Yaskawa INFORM job: TWIN_FRONT_WELD_-90ST-1_5340.JBI

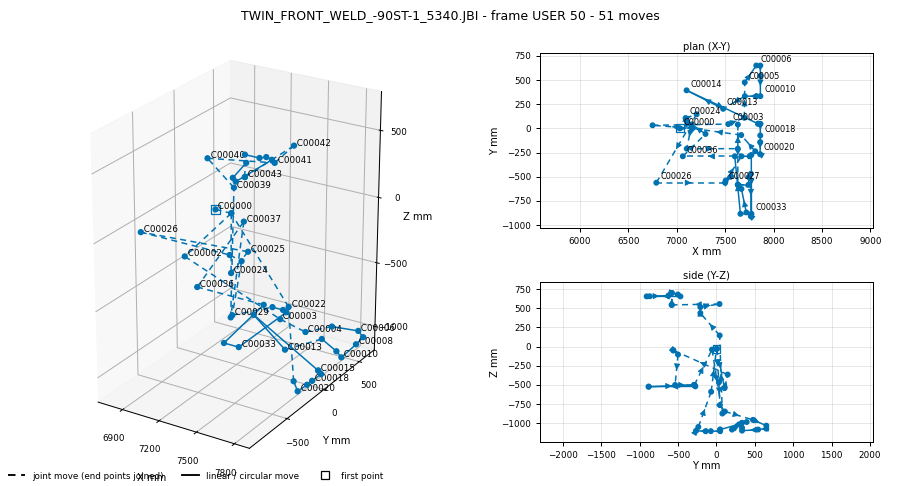
[picture p0: tool path of TWIN_FRONT_WELD_-90ST-1_5340.JBI in frame USER 50, 51 of 52 moves have a stored position in this frame; points joined in program order, loops and branches not executed]
/JOB
//NAME TWIN_FRONT_WELD_-90ST-1_5340
///FOLDERNAME 02-SKRZYNIE_JOBS
//POS
///NPOS 52,52,0,8,0,0
///USER 50
///TOOL 0
///POSTYPE USER
///RECTAN
///RCONF 0,0,1,0,0,0,0,0,0,0,0,0,0,0,0,0,0,0,0,0,0,0,0,0
C00000=7029.164,0.308,-30.113,-0.0036,-53.6521,0.0034
C00001=7158.107,0.312,-30.113,0.0036,-53.6521,-0.0034
///RCONF 1,0,1,0,0,0,0,0,0,0,0,0,0,0,0,0,0,0,0,0,0,0,0,0
C00002=6749.002,31.739,-465.549,-15.1595,35.6819,145.6807
///RCONF 1,0,0,0,0,0,0,0,0,0,0,0,0,0,0,0,0,0,0,0,0,0,0,0
C00003=7531.423,44.323,-762.797,-8.7291,34.6461,164.2133
C00004=7698.038,109.341,-845.576,-15.9625,40.0165,157.0814
C00005=7701.880,475.670,-954.346,-13.0495,30.7936,159.1476
C00006=7821.278,649.645,-1029.983,-23.6743,36.9906,149.9805
C00007=7862.724,649.337,-1069.296,-23.6733,36.9909,149.9831
C00008=7864.081,542.033,-1080.239,-23.6771,36.9818,149.9803
C00009=7863.681,455.675,-1087.596,-23.6808,36.9789,149.9684
C00010=7863.526,332.886,-1094.548,-23.6820,36.9781,149.9731
C00011=7822.668,332.804,-1057.389,-23.6776,36.9789,149.9852
C00012=7702.743,332.795,-992.444,-23.6771,36.9773,149.9828
C00013=7478.605,202.215,-1080.996,-5.5877,19.7754,112.8961
C00014=7100.516,393.258,-982.274,31.5072,20.3423,57.1288
///RCONF 0,0,0,0,0,0,0,0,0,0,0,0,0,0,0,0,0,0,0,0,0,0,0,0
C00015=7840.287,47.964,-1081.198,-15.4598,43.5968,152.6291
C00016=7840.287,47.964,-1081.198,-15.4598,43.5968,152.6291
C00017=7863.996,47.345,-1101.690,-15.0733,42.7558,153.1362
C00018=7862.274,-73.558,-1101.821,-15.0685,42.7518,153.1415
C00019=7862.125,-142.007,-1102.138,-15.0642,42.7510,153.1502
C00020=7860.827,-266.961,-1097.466,-11.5759,45.8640,155.5433
C00021=7810.369,-236.945,-1047.165,-12.8910,39.7294,154.3361
C00022=7665.368,-69.314,-588.357,-56.5185,9.2692,73.1107
///RCONF 0,0,1,0,0,0,0,0,0,0,0,0,0,0,0,0,0,0,0,0,0,0,0,0
C00023=7158.107,0.312,-30.113,0.0036,-53.6521,-0.0034
///RCONF 1,0,0,0,0,0,0,0,0,0,0,0,0,0,0,0,0,0,0,0,0,0,0,0
C00024=7089.632,105.235,-540.772,34.6747,-14.1850,-36.1511
///RCONF 0,0,0,0,0,0,0,0,0,0,0,0,0,0,0,0,0,0,0,0,0,0,0,0
C00025=7204.424,145.895,-364.343,71.1061,41.6311,-75.1821
///RCONF 1,0,1,0,0,0,0,0,0,0,0,0,0,0,0,0,0,0,0,0,0,0,0,0
C00026=6787.828,-561.979,-49.248,-84.3346,30.5101,20.5434
///RCONF 0,0,1,0,1,0,0,0,0,0,0,0,0,0,0,0,0,0,0,0,0,0,0,0
C00027=7499.847,-561.979,-49.248,-84.3345,30.5096,20.5433
///RCONF 0,0,1,0,0,0,0,0,0,0,0,0,0,0,0,0,0,0,0,0,0,0,0,0
C00028=7554.743,-500.998,-104.255,54.0039,-31.4868,-103.9439
///RCONF 0,0,0,0,0,0,0,0,0,0,0,0,0,0,0,0,0,0,0,0,0,0,0,0
C00029=7504.887,-539.129,-499.841,26.1477,-33.6094,-90.8544
C00030=7668.096,-288.720,-499.869,26.1496,-33.6072,-90.8555
C00031=7751.665,-288.695,-499.888,50.2103,-29.8101,-103.4316
C00032=7769.646,-275.360,-518.298,50.1633,-29.8093,-103.3948
C00033=7771.403,-883.462,-522.090,50.1989,-29.8077,-103.4313
C00034=7657.159,-883.464,-522.091,50.1980,-29.8087,-103.4305
C00035=7598.862,-288.695,-499.888,50.2103,-29.8101,-103.4316
C00036=7061.929,-288.695,-499.888,50.2103,-29.8101,-103.4316
C00037=7296.409,-57.933,-39.561,132.2856,-81.6072,-138.1355
C00038=7103.855,76.465,-871.663,11.0010,-20.3154,-11.3718
///RCONF 1,0,1,0,0,0,0,0,0,0,0,0,0,0,0,0,0,0,0,0,0,0,0,0
C00039=7154.189,41.489,145.490,17.6136,-33.4406,-10.5318
C00040=7102.089,-209.900,436.597,-19.7303,-44.5925,9.1969
C00041=7630.528,-209.897,514.987,-19.7320,-44.5912,9.1993
C00042=7630.530,39.680,554.688,-52.1357,-35.3916,30.4208
C00043=7630.500,-582.850,542.955,-61.9434,-30.0005,35.7331
C00044=7630.491,-582.857,542.952,-61.9449,-29.9979,35.7338
C00045=7630.501,-582.856,698.927,-61.9436,-29.9977,35.7338
C00046=7740.859,-582.856,698.927,-61.9436,-29.9977,35.7338
C00047=7743.607,-503.312,679.062,-61.9419,-29.9985,35.7328
C00048=7765.899,-469.746,653.450,-60.1061,-26.9469,34.8664
C00049=7765.598,-909.634,654.025,-56.0408,-31.7443,29.4745
C00050=7718.203,-868.976,655.452,-56.0446,-31.7378,29.4783
C00051=7667.415,-626.051,664.446,-58.3119,-31.1539,31.9267
///RCONF 0,0,0,0,0,0,0,0,0,0,0,0,0,0,0,0,0,0,0,0,0,0,0,0
BC00000=5214.746
BC00001=5343.689
BC00002=5343.689
BC00003=6178.800
BC00004=6495.017
BC00005=6648.627
BC00006=6688.143
BC00007=6688.143
BC00008=6688.143
BC00009=6688.144
BC00010=6688.144
BC00011=6688.143
BC00012=6688.143
BC00013=6688.144
BC00014=6688.143
BC00015=6686.021
BC00016=6686.021
BC00017=6686.021
BC00018=6686.034
BC00019=6686.047
BC00020=6686.060
BC00021=6686.021
BC00022=6015.470
BC00023=5343.689
BC00024=5388.459
BC00025=5388.459
BC00026=5388.459
BC00027=6100.478
BC00028=6100.478
BC00029=6331.805
BC00030=6331.805
BC00031=6331.805
BC00032=6331.785
BC00033=6331.785
BC00034=6331.785
BC00035=6179.002
BC00036=5642.069
BC00037=5642.069
BC00038=5642.069
BC00039=5642.069
BC00040=5642.069
BC00041=6170.513
BC00042=6170.513
BC00043=6170.513
BC00044=6302.692
BC00045=6302.692
BC00046=6413.050
BC00047=6413.050
BC00048=6413.056
BC00049=6735.412
BC00050=6672.519
BC00051=6394.301
///POSTYPE BASE
P00021=6.550,-0.003,-5.735,0.0000,0.0000,0.0000
P00022=5.943,-0.018,-6.388,0.0000,0.0000,0.0000
P00023=7.025,-0.019,-7.168,0.0000,0.0000,0.0000
P00024=5.926,-0.047,-4.777,0.0000,0.0000,0.0000
P00501=-2.026,0.009,3.534,0.0000,0.0000,0.0000
///RCONF 1,0,0,0,0,0,0,0,0,0,0,0,0,0,0,0,0,0,0,0,0,0,0,0
P00502=-2.023,0.001,1.732,0.0000,0.0000,0.0000
P00503=0.138,-0.044,1.539,0.0000,0.0000,0.0000
P00504=-0.309,-0.010,1.636,0.0000,0.0000,0.0000
//INST
///DATE 2024/12/18 13:42
///ATTR SC,RW,RJ
////FRAME USER 50
///GROUP1 RB1,BS1
NOP
MOVJ C00000 BC00000 VJ=50.00
MOVJ C00001 BC00001 VJ=50.00
MOVJ C00002 BC00002 VJ=50.00
MOVJ C00003 BC00003 VJ=50.00
MOVJ C00004 BC00004 VJ=50.00
MOVJ C00005 BC00005 VJ=50.00
'::::::::::::::::::::::::::::::::
'W56
'::::::::::::::::::::::::::::::::
MOVL C00006 BC00006 V=500.0
SFTON P0501
MACRO1 MJ#(0) ARGF14
MOVL C00007 BC00007 V=166.7 PL=0
ARCON
MOVC C00008 BC00008 V=9.5
SFTOF
SFTON P0502
MOVC C00009 BC00009 V=9.5
MOVC C00010 BC00010 V=9.5
ARCOF
MOVL C00011 BC00011 V=166.7
SFTOF
MOVL C00012 BC00012 V=166.7
MOVJ C00013 BC00013 VJ=30.00
MOVL C00014 BC00014 V=166.7
MOVL C00015 BC00015 V=166.7
'::::::::::::::::::::::::::::::::
'W21
'::::::::::::::::::::::::::::::::
MOVL C00016 BC00016 V=166.7
SFTON P0503
MACRO1 MJ#(0) ARGF14
MOVL C00017 BC00017 V=166.7 PL=0
ARCON
MOVL C00018 BC00018 V=9.5
SFTOF
SFTON P0504
MOVL C00019 BC00019 V=9.5
MOVL C00020 BC00020 V=9.5
ARCOF
MOVL C00021 BC00021 V=250.0
SFTOF
MOVJ C00022 BC00022 VJ=30.00
MOVJ C00023 BC00023 VJ=50.00
MOVJ C00024 BC00024 VJ=50.00
MOVJ C00025 BC00025 VJ=50.00
MOVJ C00026 BC00026 VJ=50.00
MOVJ C00027 BC00027 VJ=50.00
MOVJ C00028 BC00028 VJ=50.00
MOVJ C00029 BC00029 VJ=50.00
MOVJ C00030 BC00030 VJ=50.00
MOVL C00031 BC00031 V=166.7
MACRO1 MJ#(0) ARGF9
SFTON P0021
MOVL C00032 BC00032 V=166.7
ARCON
SFTON P0022
MOVL C00033 BC00033 V=9.2
ARCOF
MOVL C00034 BC00034 V=166.7
SFTOF
MOVL C00035 BC00035 V=166.7
MOVJ C00036 BC00036 VJ=50.00
MOVJ C00037 BC00037 VJ=50.00
MOVJ C00038 BC00038 VJ=50.00
MOVJ C00039 BC00039 VJ=50.00
MOVJ C00040 BC00040 VJ=50.00
MOVJ C00041 BC00041 VJ=50.00
MOVJ C00042 BC00042 VJ=50.00
MOVJ C00043 BC00043 VJ=50.00
MOVJ C00044 BC00044 VJ=50.00
MOVJ C00045 BC00045 VJ=50.00
MOVL C00046 BC00046 V=166.7
MOVL C00047 BC00047 V=166.7
SFTON P0023
MOVL C00048 BC00048 V=166.7 PL=0
ARCON
SFTON P0024
MOVL C00049 BC00049 V=9.2
ARCOF
MOVL C00050 BC00050 V=166.7
SFTOF
MOVL C00051 BC00051 V=166.7
END
